# EPICS autosave request: dxp/tags/R2-4/iocBoot/iocXMAP/auto_settings4.req
file "simple_mca_settings.req",         P=dxpXMAP:med:, M=mca1
file "dxp_settings.req",                P=dxpXMAP:med:, R=dxp1
file "simple_mca_settings.req",         P=dxpXMAP:med:, M=mca2
file "dxp_settings.req",                P=dxpXMAP:med:, R=dxp2
file "simple_mca_settings.req",         P=dxpXMAP:med:, M=mca3
file "dxp_settings.req",                P=dxpXMAP:med:, R=dxp3
file "simple_mca_settings.req",         P=dxpXMAP:med:, M=mca4
file "dxp_settings.req",                P=dxpXMAP:med:, R=dxp4
